FUNCTION f_MQTTPUB : BOOL
VAR_INPUT
	
		MqttClient: FB_IotMqttClient;		
		sTopic : STRING;
		sValue : STRING;

END_VAR
VAR
	sPayloadPub: STRING;
END_VAR

        MqttClient.Publish(    sTopic:= sTopic, 
			                   pPayload:= ADR(sValue), nPayloadSize:= LEN2(ADR(sValue))+1, 
                               eQoS:= TcIotMqttQos.AtMostOnceDelivery, bRetain:= FALSE, bQueue:= FALSE );

END_FUNCTION

(* stored: Version 1.1.0.1, ProductVersion 3.1.4024.12
   POU f_MQTTPUB: Id {60ac643d-7601-4c31-8331-24ab4e3f3f40}, SpecialFunc None *)
